INTERFACE I_Skill_RoboterErweitert

METHOD M_Reset : BOOL
VAR_INPUT
END_VAR
END_METHOD

METHOD M_Start : BOOL
VAR_INPUT
END_VAR
END_METHOD

METHOD M_Stop : BOOL
VAR_INPUT
END_VAR
END_METHOD

PROPERTY P_Erreicht : sKraftVariablen
SET
END_SET
END_PROPERTY

PROPERTY P_Limit : sKraftVariablen
SET
END_SET
END_PROPERTY

PROPERTY P_RobotParam : sRoboterProzessVariablen
SET
END_SET
END_PROPERTY

PROPERTY P_State : eSkillState
GET
END_GET
END_PROPERTY

END_INTERFACE

(* stored: Version 1.1.0.1
   Itf I_Skill_RoboterErweitert: Id {e2d1cd4d-0af3-4bdf-a370-2bb2a0007c52}
   Method M_Reset: Id {b6ae5578-e81b-4948-b312-0c318809c1a1}
   Method M_Start: Id {b6618813-d193-4b86-a2e9-1449f0a7f8b3}
   Method M_Stop: Id {7674e0b9-c88f-4588-b850-020e9f541814}
   Property P_Erreicht: Id {d6f9089f-3c67-49dd-8b6a-3d7c5b7d3083}
   Set Set: Id {80788c3c-21e3-4396-b662-e3fd0325bd45}
   Property P_Limit: Id {631cb066-0c7c-4b39-a9bd-28dbd6482768}
   Set Set: Id {bad53743-5c4e-4d00-b4f5-0a3573daa2fb}
   Property P_RobotParam: Id {c1f9be14-e652-476d-91a4-fce89d221794}
   Set Set: Id {97851a4a-6624-4bd3-a0d4-54b8c92d2ac3}
   Property P_State: Id {55efd3f7-15fa-4776-bbf3-efdf75362085}
   Get Get: Id {f4c65372-93b7-4b2f-a55e-a642f1d854ed} *)
